FUNCTION_BLOCK disponivelAuto (* Extracted Composite Function Block Type *)
  (* Standard: 61499-2 *)
  (* Version 24/02/2026 *)
  PACKAGE Hidryco.HidrycoLib;
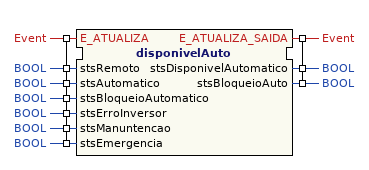
  EVENT_INPUT
    E_ATUALIZA WITH stsRemoto, stsAutomatico, stsBloqueioAutomatico, stsErroInversor, stsManuntencao, stsEmergencia;
  END_EVENT
  EVENT_OUTPUT
    E_ATUALIZA_SAIDA WITH stsBloqueioAuto, stsDisponivelAutomatico; (* Execution Confirmation *)
  END_EVENT
  VAR_INPUT
    stsRemoto : BOOL; (* Argument *)
    stsAutomatico : BOOL; (* Argument *)
    stsBloqueioAutomatico : BOOL; (* Argument *)
    stsErroInversor : BOOL; (* Argument *)
    stsManuntencao : BOOL; (* Argument *)
    stsEmergencia : BOOL; (* Argument *)
  END_VAR
  VAR_OUTPUT
    stsDisponivelAutomatico : BOOL; (* Result: IN1 AND IN2 AND ... *)
    stsBloqueioAuto : BOOL; (* Result: IN1 OR IN2 OR ... *)
  END_VAR
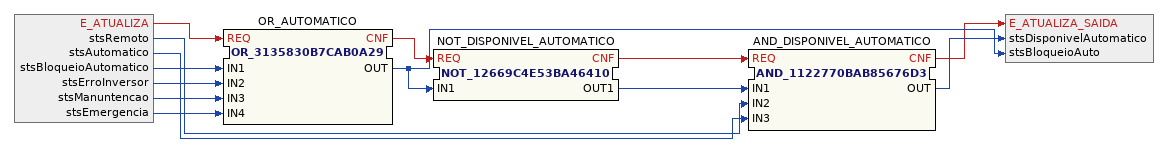
  FBS
    OR_AUTOMATICO : OR_3135830B7CAB0A29; {SET_ATTRIBUTE(Configuration.GenericFBType.InterfaceParams, Runtime.Standard#CNT:=4)}
    NOT_DISPONIVEL_AUTOMATICO : NOT_12669C4E53BA46410; {SET_ATTRIBUTE(Configuration.GenericFBType.InterfaceParams, Runtime.Standard#CNT:=1)}
    AND_DISPONIVEL_AUTOMATICO : AND_1122770BAB85676D3; {SET_ATTRIBUTE(Configuration.GenericFBType.InterfaceParams, Runtime.Standard#CNT:=3)}
  END_FBS
  EVENT_CONNECTIONS
    NOT_DISPONIVEL_AUTOMATICO.CNF TO AND_DISPONIVEL_AUTOMATICO.REQ;
    OR_AUTOMATICO.CNF TO NOT_DISPONIVEL_AUTOMATICO.REQ;
    AND_DISPONIVEL_AUTOMATICO.CNF TO E_ATUALIZA_SAIDA;
    E_ATUALIZA TO OR_AUTOMATICO.REQ;
  END_CONNECTIONS
  DATA_CONNECTIONS
    NOT_DISPONIVEL_AUTOMATICO.OUT1 TO AND_DISPONIVEL_AUTOMATICO.IN1;
    OR_AUTOMATICO.OUT TO NOT_DISPONIVEL_AUTOMATICO.IN1;
    stsRemoto TO AND_DISPONIVEL_AUTOMATICO.IN2;
    stsAutomatico TO AND_DISPONIVEL_AUTOMATICO.IN3;
    AND_DISPONIVEL_AUTOMATICO.OUT TO stsDisponivelAutomatico;
    stsBloqueioAutomatico TO OR_AUTOMATICO.IN1;
    stsErroInversor TO OR_AUTOMATICO.IN2;
    stsManuntencao TO OR_AUTOMATICO.IN3;
    stsEmergencia TO OR_AUTOMATICO.IN4;
    OR_AUTOMATICO.OUT TO stsBloqueioAuto;
  END_CONNECTIONS
END_FUNCTION_BLOCK
